TYPE Vision_Outputs_typ:
STRUCT
	Inspect AT %Q*: BOOL;
END_STRUCT
END_TYPE

(* stored: Version 1.1.0.1, ProductVersion 3.1.4024.12
   DUT Vision_Outputs_typ: Id {609b1b23-392a-01dd-3273-6bcf9e069b20} *)
